// TIA Portal V19 export
FUNCTION "FC_WT_MANAGER" : Void   // FC40, STL
TITLE = WT-Manager
{ S7_Optimized_Access := 'FALSE' }
AUTHOR : MS
// Verwaltung der Wt an Auf- und Ausgabestationen
// Technologiezuweisung
// stored: AutoNumber false
   VAR_TEMP
      FW_kommt : Bool;
      FW_in_Pos : Bool;
      Ziel_FW : Bool;
      STAND_POS : Byte;
      Param : DWord;
      AutoDelete : Bool;
      DeleteAll : Bool;
      Anforderung_QF : Bool;
      Sperre_TW : Bool;
   END_VAR
BEGIN

NETWORK
TITLE = Technologie
// Zuweisung on Technologien
//Programme laden

      CALL  "FC_Rez_to_DB45";

      CALL  "FC_AEND_WT";


NETWORK
TITLE = Check Querförderer
      A     "DI_QF_WR02_03".Zst.Req_WR02_In;
      O     "DI_QF_WR02_03".Zst.Req_WR03_In;
      O     "DI_QF_WR02_03".Zst.Req_WR02_Out;
      O     "DI_QF_WR02_03".Zst.Req_WR03_Out;
      O     "DI_QF_WR02_03".Out.WR02_einfahren;
      O     "DI_QF_WR02_03".Out.WR02_ausfahren;
      O     "DI_QF_WR02_03".Out.WR03_einfahren;
      O     "DI_QF_WR02_03".Out.WR03_ausfahren;
      =     #Anforderung_QF;

      A     "DI_QF_WR02_03".Zst.Req_WR02_In;
      O     "DI_QF_WR02_03".Zst.Req_WR03_In;
      O     "DI_QF_WR02_03".Zst.Req_WR02_Out;
      O     "DI_QF_WR02_03".Zst.Req_WR03_Out;
      A     "DI_QF_WR02_03".Zst.TW_sicher;
      O     "DI_QF_WR02_03".Out.WR02_einfahren;
      O     "DI_QF_WR02_03".Out.WR02_ausfahren;
      O     "DI_QF_WR02_03".Out.WR03_einfahren;
      O     "DI_QF_WR02_03".Out.WR03_ausfahren;
      =     #Sperre_TW;


NETWORK
TITLE = Beladestände
      A     "DB_ANLAGE".BA.Simulation;
      =     #AutoDelete;
      SET;
      =     #DeleteAll;

//-----------------------------
//Beladestand 1
//-----------------------------
      CALL  "FC_Beladen"
      ( Stand_Nr       := 1,
        E_Belegt       := "DB_BE_Stand".Stand[1].IN_Belegt,
        E_S_innen      := "DB_BE_Stand".Stand[1].IN_innen,
        E_S_aussen     := "DB_BE_Stand".Stand[1].IN_aussen,
        E_S_verriegelt := "DB_BE_Stand".Stand[1].verriegelt,
        E_Freigabe     := "DB_BE_Stand".Stand[1].IN_Freigabe,
        Auto_Delete    := #AutoDelete,
        ext_Delete     := FALSE,
        Del_All        := #DeleteAll,
        Afg_WT_Nr      := false,
        Del_count      := 5
      );

      A     "DB_BE_Stand".Stand[1].OUT_Sperre_in;
      O     #Anforderung_QF;
      =     "DB_POS".POS[25].notFG_in;

// GO links
      L     "DB_POS".POS[27].next_WT;
      L     0;
      <>I;
      S     "DB_POS".POS[25].notFG_in;

      A     "DB_BE_Stand".Stand[1].OUT_Sperre_FW;
      O     #Sperre_TW;
      O(;
      A     "DI_FW_1".ZST.Oben_li;
      A(;
      A     "DB_BE_Stand".Stand[1].IN_Belegt;
      O     "DB_POS".POS[25].belegt;
      AN    "DB_BE_Stand".Stand[1].IN_aussen;
      );
      O;
      A     "DI_FW_1".ZST.Oben_re;
      A(;
      A     "DB_BE_Stand".Stand[2].IN_Belegt;
      O     "DB_POS".POS[26].belegt;
      AN    "DB_BE_Stand".Stand[2].IN_aussen;
      );
      );
      =     "DB_POS".POS[25].Sperre_FW;

      A     "DB_BE_Stand".Stand[1].OUT_Sperre_out;
      O     #Anforderung_QF;
      =     "DB_POS".POS[25].notFG_out;

//-----------------------------
//Beladestand 2
//-----------------------------
      CALL  "FC_Beladen"
      ( Stand_Nr       := 2,
        E_Belegt       := "DB_BE_Stand".Stand[2].IN_Belegt,
        E_S_innen      := "DB_BE_Stand".Stand[2].IN_innen,
        E_S_aussen     := "DB_BE_Stand".Stand[2].IN_aussen,
        E_S_verriegelt := "DB_BE_Stand".Stand[2].verriegelt,
        E_Freigabe     := "DB_BE_Stand".Stand[2].IN_Freigabe,
        Auto_Delete    := #AutoDelete,
        ext_Delete     := FALSE,
        Del_All        := #DeleteAll,
        Afg_WT_Nr      := false,
        Del_count      := 5
      );

      A     "DB_BE_Stand".Stand[2].OUT_Sperre_in;
      O     #Anforderung_QF;
      =     "DB_POS".POS[26].notFG_in;
// GO rechts
      L     "DB_POS".POS[28].next_WT;
      L     0;
      <>I;
      S     "DB_POS".POS[26].notFG_in;

      A     "DB_BE_Stand".Stand[2].OUT_Sperre_out;
      O     #Anforderung_QF;
      =     "DB_POS".POS[26].notFG_out;

//-----------------------------
//Beladestand 3 (GO links)
//-----------------------------
      CALL  "FC_Beladen"
      ( Stand_Nr       := 3,
        E_Belegt       := "DB_BE_Stand".Stand[3].IN_Belegt,
        E_S_innen      := "DB_BE_Stand".Stand[3].IN_innen,
        E_S_aussen     := "DB_BE_Stand".Stand[3].IN_aussen,
        E_S_verriegelt := "DB_BE_Stand".Stand[3].verriegelt,
        E_Freigabe     := "DB_BE_Stand".Stand[3].IN_Freigabe,
        Auto_Delete    := #AutoDelete,
        ext_Delete     := FALSE,
        Del_All        := #DeleteAll,
        Afg_WT_Nr      := false,
        Del_count      := 5
      );

      A     "DB_BE_Stand".Stand[3].OUT_Sperre_in;
      O     #Anforderung_QF;
      =     "DB_POS".POS[27].notFG_in;

//KS links
      L     "DB_POS".POS[25].next_WT;
      L     0;
      <>I;
      O(;
      L     "DB_POS".POS[29].next_WT;
      <>I;
      );
      O(;
      A     "DB_BE_Stand".Stand[1].IN_Belegt;
      A     "DB_BE_Stand".Stand[1].IN_innen;
      );
      O(;
      A     "DB_BE_Stand".Stand[5].IN_Belegt;
      A     "DB_BE_Stand".Stand[5].IN_innen;
      );
      S     "DB_POS".POS[27].notFG_in;

      A     "DB_BE_Stand".Stand[3].OUT_Sperre_out;
      O     #Anforderung_QF;
      =     "DB_POS".POS[27].notFG_out;

//-----------------------------
//Beladestand 4 (GO rechts)
//-----------------------------
      CALL  "FC_Beladen"
      ( Stand_Nr       := 4,
        E_Belegt       := "DB_BE_Stand".Stand[4].IN_Belegt,
        E_S_innen      := "DB_BE_Stand".Stand[4].IN_innen,
        E_S_aussen     := "DB_BE_Stand".Stand[4].IN_aussen,
        E_S_verriegelt := "DB_BE_Stand".Stand[4].verriegelt,
        E_Freigabe     := "DB_BE_Stand".Stand[4].IN_Freigabe,
        Auto_Delete    := #AutoDelete,
        ext_Delete     := FALSE,
        Del_All        := #DeleteAll,
        Afg_WT_Nr      := false,
        Del_count      := 5
      );

      A     "DB_BE_Stand".Stand[4].OUT_Sperre_in;
      O     #Anforderung_QF;
      =     "DB_POS".POS[28].notFG_in;
//KS rechts
      L     "DB_POS".POS[26].next_WT;
      L     0;
      <>I;
      O(;
      L     "DB_POS".POS[30].next_WT;
      <>I;
      );
      O(;
      A     "DB_BE_Stand".Stand[2].IN_Belegt;
      A     "DB_BE_Stand".Stand[2].IN_innen;
      );
      O(;
      A     "DB_BE_Stand".Stand[6].IN_Belegt;
      A     "DB_BE_Stand".Stand[6].IN_innen;
      );
      S     "DB_POS".POS[28].notFG_in;

      A     "DB_BE_Stand".Stand[4].OUT_Sperre_out;
      O     #Anforderung_QF;
      =     "DB_POS".POS[28].notFG_out;

//-------------------------------
//Beladestand 5 (KS hinten links)
//-------------------------------
      CALL  "FC_Beladen"
      ( Stand_Nr       := 5,
        E_Belegt       := "DB_BE_Stand".Stand[5].IN_Belegt,
        E_S_innen      := "DB_BE_Stand".Stand[5].IN_innen,
        E_S_aussen     := "DB_BE_Stand".Stand[5].IN_aussen,
        E_S_verriegelt := "DB_BE_Stand".Stand[5].verriegelt,
        E_Freigabe     := "DB_BE_Stand".Stand[5].IN_Freigabe,
        Auto_Delete    := #AutoDelete,
        ext_Delete     := FALSE,
        Del_All        := #DeleteAll,
        Afg_WT_Nr      := false,
        Del_count      := 5
      );

      L     "DB_POS".POS[25].next_WT;
      L     0;
      <>I;
      O     "DB_BE_Stand".Stand[1].IN_Belegt;
      AN    "DB_BE_Stand".Stand[1].IN_aussen;
      O     "DB_BE_Stand".Stand[5].OUT_Sperre_in;
      O     #Anforderung_QF;
      =     "DB_POS".POS[29].notFG_in;
// GO links
      L     "DB_POS".POS[27].next_WT;
      L     0;
      <>I;
      S     "DB_POS".POS[29].notFG_in;

      A     "DB_BE_Stand".Stand[5].OUT_Sperre_FW;
      O(;
      A     "DB_POS".POS[29].FW_in_POS;
      A(;
      A     "DI_FW_1".ZST.Oben_li;
      A(;
      A     "DB_BE_Stand".Stand[1].IN_Belegt;
      O     "DB_POS".POS[25].belegt;
      AN    "DB_BE_Stand".Stand[1].IN_aussen;
      );
      O;
      A     "DI_FW_1".ZST.Oben_re;
      A(;
      A     "DB_BE_Stand".Stand[2].IN_Belegt;
      O     "DB_POS".POS[26].belegt;
      AN    "DB_BE_Stand".Stand[2].IN_aussen;
      );
      );
      );
      O     #Sperre_TW;
      =     "DB_POS".POS[29].Sperre_FW;

      L     "DB_POS".POS[25].next_WT;
      L     0;
      <>I;
      O     "DB_BE_Stand".Stand[1].IN_Belegt;
      AN    "DB_BE_Stand".Stand[1].IN_aussen;
      O     "DB_BE_Stand".Stand[5].OUT_Sperre_out;
      O     #Anforderung_QF;
      =     "DB_POS".POS[29].notFG_out;

//--------------------------------
//Beladestand 6 (KS hinten rechts)
//--------------------------------
      CALL  "FC_Beladen"
      ( Stand_Nr       := 6,
        E_Belegt       := "DB_BE_Stand".Stand[6].IN_Belegt,
        E_S_innen      := "DB_BE_Stand".Stand[6].IN_innen,
        E_S_aussen     := "DB_BE_Stand".Stand[6].IN_aussen,
        E_S_verriegelt := "DB_BE_Stand".Stand[6].verriegelt,
        E_Freigabe     := "DB_BE_Stand".Stand[6].IN_Freigabe,
        Auto_Delete    := #AutoDelete,
        ext_Delete     := FALSE,
        Del_All        := #DeleteAll,
        Afg_WT_Nr      := false,
        Del_count      := 5
      );


      L     "DB_POS".POS[26].next_WT;
      L     0;
      <>I;
      O     "DB_BE_Stand".Stand[2].IN_Belegt;
      AN    "DB_BE_Stand".Stand[2].IN_aussen;
      O     "DB_BE_Stand".Stand[6].OUT_Sperre_in;
      O     #Anforderung_QF;
      =     "DB_POS".POS[30].notFG_in;
// GO rechts
      L     "DB_POS".POS[28].next_WT;
      L     0;
      <>I;
      S     "DB_POS".POS[30].notFG_in;

      L     "DB_POS".POS[26].next_WT;
      L     0;
      <>I;
      O     "DB_BE_Stand".Stand[2].IN_Belegt;
      AN    "DB_BE_Stand".Stand[2].IN_aussen;
      O     "DB_BE_Stand".Stand[6].OUT_Sperre_out;
      O     #Anforderung_QF;
      =     "DB_POS".POS[30].notFG_out;

END_FUNCTION
